FUNCTION fcEvalConitinuos : BOOL
VAR_INPUT
	Val : REAL;
END_VAR
VAR_IN_OUT
	Data : stContinuosValueData;
END_VAR

Data.Measured := Val;
fcEvalConitinuos := (Data.Mininum <= Data.Measured AND Data.Measured <= Data.Maximum);

END_FUNCTION

(* stored: Version 1.1.0.1, ProductVersion 3.1.4024.2
   POU fcEvalConitinuos: Id {e63b02de-1ad8-4dfc-8e0c-28ef7017ed74}, SpecialFunc None *)
